Yaskawa INFORM job: HOME_B.JBI

/JOB
//NAME HOME_B
///FOLDERNAME MASTER
//POS
///NPOS 0,0,0,0,0,1
///TOOL 0
///POSTYPE PULSE
///PULSE
EX00050=-200
//INST
///DATE 2021/10/29 11:48
///ATTR SC,RO
///GROUP1 ST1
NOP
'*******************************
'THIS JOB HOMES POSITIONER SIDE
'B TO THE ROBOT, SIDE A TO LOAD
'WITHOUT AFFECTING THE TOOLING.
'********************************
MOVJ EX050 VJ=5.00
END
